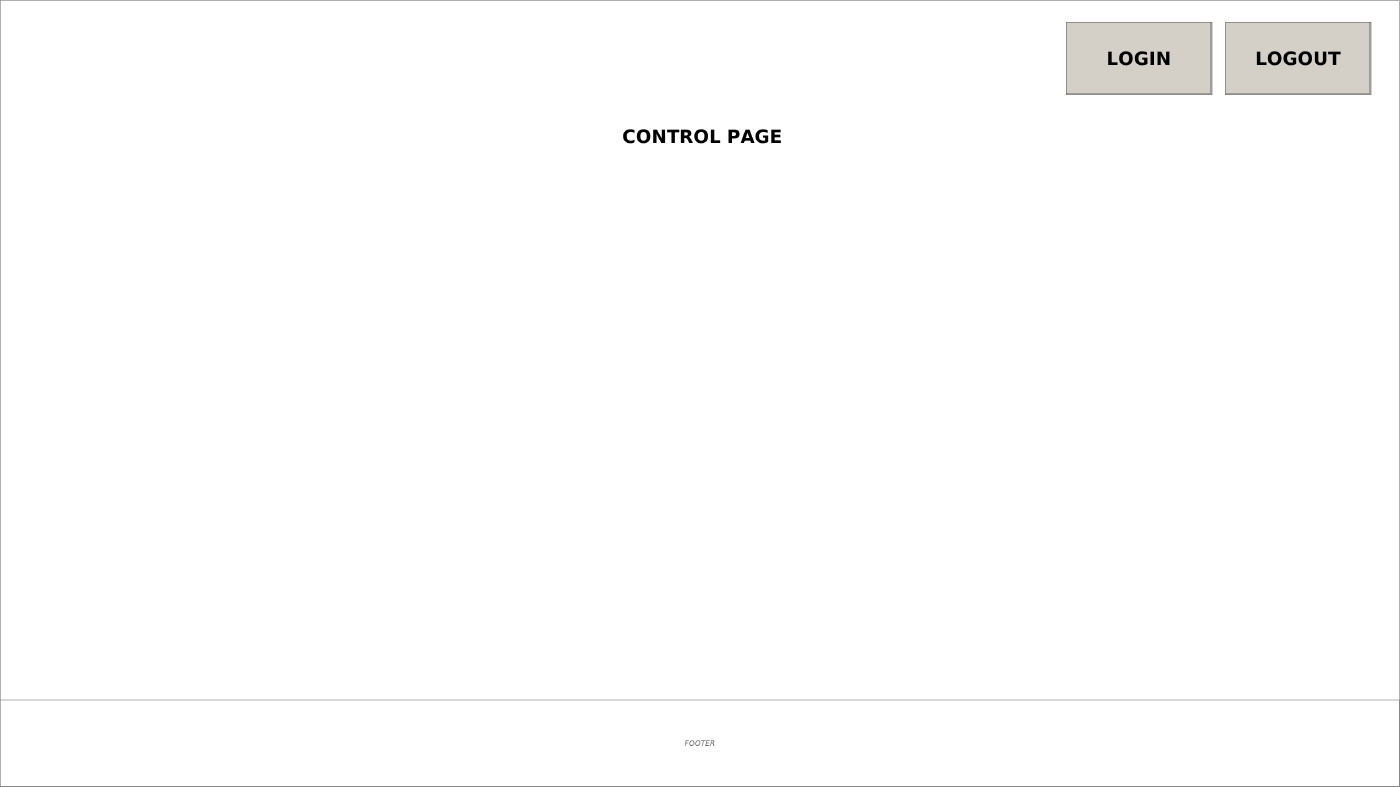
VISUALIZATION PAGE_CONTROL  // 1920x1080, background image ImagePool.Grey_Gradient
    Button (1462,30 200x100), "LOGIN"
        OnMouseClick: VisuUserMgmt Type=Login
    Button (1680,30 200x100), "LOGOUT"
        OnMouseClick: VisuUserMgmt Type=Logout
    Frame (0,960 1920x120)
        shows FOOTER()
    Label (728,129 470x116), "CONTROL PAGE"
END_VISUALIZATION

(* stored: Version 1.1.0.1, ProductVersion 3.1.4024.12
   Visu PAGE_CONTROL: Id {73a3a3b3-099b-4346-9f4c-0fff8546ac87} *)
